FUNCTION_BLOCK FB_Opcpa
VAR_INPUT
	nOpcpaVoltageRaw : INT;
	bAmphosOn : BOOL;
END_VAR
VAR_IN_OUT
	stSetpoints : ST_LaserSetpoints;
END_VAR
VAR_OUTPUT
	fOpcpaVoltage : LREAL;
	bError : BOOL;
END_VAR
VAR
END_VAR

fOpcpaVoltage := F_Scale(
	fRawData := nOpcpaVoltageRaw,
	fRawDataLowerOffLimit := GVL_EL3174.fRawLowerLimit,
	fRawDataUpperOffLimit := GVL_EL3174.fRawUpperLimit,
	fScaleDataLowerOffLimit := GVL_EL3174.fScaleLowerLimit,
	fScaleDataUpperOffLimit := GVL_EL3174.fScaleUpperLimit);
	
IF  bAmphosOn AND fOpcpaVoltage < stSetpoints.nMinNominalVoltage THEN
	bError := TRUE;
END_IF

METHOD Reset : BOOL
VAR_INPUT
END_VAR
bError := FALSE;
END_METHOD

END_FUNCTION_BLOCK

(* stored: Version 1.1.0.1, ProductVersion 3.1.4020.14
   POU FB_Opcpa: Id {b09b705a-b75a-44ab-aab6-38306d5c5f30}, SpecialFunc None
   Method Reset: Id {1c7a9fd1-6742-422e-8400-0035b7297bfe} *)
